FUNCTION_BLOCK A2X_SUBSCRIBE_2 (* Subscribe to a PUBLISH_2 Block and buffer both received BOOLs with a D_FF each, delivered on an A2X adapter Plug *)
  (* Standard: 61499-2; Description: Copyright (c) 2026 HR Agrartechnik GmbH This program and the accompanying materials are made available under the terms of the Eclipse Public License 2.0 which is available at https://www.eclipse.org/legal/epl-2.0/ SPDX-License-Identifier: EPL-2.0 *)
  (* Version 1.0, 2026-09-05, Franz Höpfinger, HR Agrartechnik GmbH, initial API and implementation and/or initial documentation *)
  PACKAGE adapter::net;
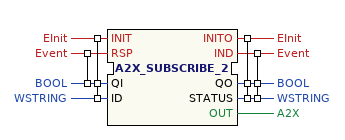
  EVENT_INPUT
    INIT : EInit WITH QI, ID; (* Initialization *)
    RSP WITH QI; (* Response to the received data *)
  END_EVENT
  EVENT_OUTPUT
    INITO : EInit WITH QO, STATUS; (* Initialization Confirm *)
    IND WITH QO, STATUS; (* New data available *)
  END_EVENT
  VAR_INPUT
    QI : BOOL;
    ID : WSTRING;
  END_VAR
  VAR_OUTPUT
    QO : BOOL;
    STATUS : WSTRING;
  END_VAR
  PLUGS
    OUT : adapter::types::unidirectional::A2X; (* Buffered received UP/DOWN BOOLs *)
  END_PLUGS
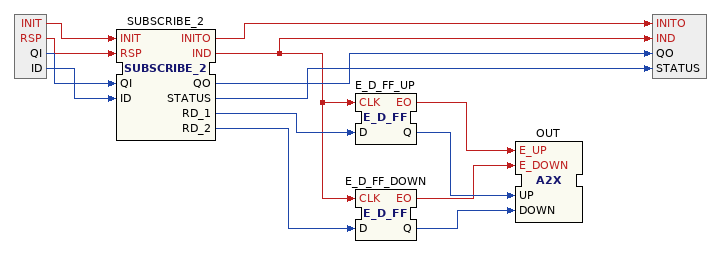
  FBS
    SUBSCRIBE_2 : iec61499::net::SUBSCRIBE_2;
    E_D_FF_UP : iec61499::events::E_D_FF;
    E_D_FF_DOWN : iec61499::events::E_D_FF;
  END_FBS
  EVENT_CONNECTIONS
    INIT TO SUBSCRIBE_2.INIT;
    RSP TO SUBSCRIBE_2.RSP;
    SUBSCRIBE_2.INITO TO INITO;
    SUBSCRIBE_2.IND TO E_D_FF_UP.CLK;
    SUBSCRIBE_2.IND TO E_D_FF_DOWN.CLK;
    E_D_FF_UP.EO TO OUT.E_UP;
    E_D_FF_DOWN.EO TO OUT.E_DOWN;
    SUBSCRIBE_2.IND TO IND;
  END_CONNECTIONS
  DATA_CONNECTIONS
    QI TO SUBSCRIBE_2.QI;
    ID TO SUBSCRIBE_2.ID;
    SUBSCRIBE_2.QO TO QO;
    SUBSCRIBE_2.STATUS TO STATUS;
    SUBSCRIBE_2.RD_1 TO E_D_FF_UP.D;
    SUBSCRIBE_2.RD_2 TO E_D_FF_DOWN.D;
    E_D_FF_UP.Q TO OUT.UP;
    E_D_FF_DOWN.Q TO OUT.DOWN;
  END_CONNECTIONS
END_FUNCTION_BLOCK
